FUNCTION_BLOCK FB_CAM
VAR_INPUT
	bAruco 	: BOOL;
	bProxi	: BOOL;
END_VAR
VAR_OUTPUT
	TAruco 			: ARRAY [0..10] OF INT;
	usiProximite 	: USINT;
END_VAR

//author: Alec Horth

//gestion des fonctionnalités de la caméra
// voir GVL "G_CAM" pour plus de détails d'implémentation
G_CAM.RUN_ARUCO := bAruco;
IF bAruco THEN
	TAruco := G_CAM.tag_aruco;
END_IF

G_CAM.RUN_STEREO := bProxi;
IF bProxi THEN
	usiProximite := G_CAM.proximite;
END_IF

END_FUNCTION_BLOCK

(* stored: Version 1.1.0.1, ProductVersion 3.1.4024.11
   POU FB_CAM: Id {bbef3e1a-0090-4306-af96-8827d31b9c29}, SpecialFunc None *)
